FUNCTION_BLOCK TWO_POS_AXIS (* Composite Function Block Type *)
  (* Standard: 61499-2 *)
  (* Version 0.0, 4/29/2023, Dmitrii, Flexbridge AB, template *)
  PACKAGE UAO.Hackathon;
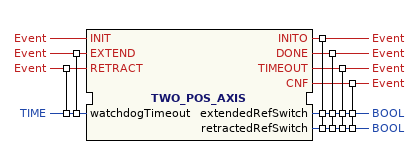
  EVENT_INPUT
    INIT; (* Initialization Request *)
    EXTEND WITH watchdogTimeout; (* Normal Execution Request *)
    RETRACT WITH watchdogTimeout;
  END_EVENT
  EVENT_OUTPUT
    INITO WITH extendedRefSwitch, retractedRefSwitch; (* Initialization Confirm *)
    DONE WITH retractedRefSwitch, extendedRefSwitch; (* Execution Confirmation *)
    TIMEOUT WITH retractedRefSwitch, extendedRefSwitch;
    CNF WITH extendedRefSwitch, retractedRefSwitch; (* Confirmation of an explicit or implicit data read request *)
  END_EVENT
  VAR_INPUT
    watchdogTimeout : TIME; (* Delay Time *)
  END_VAR
  VAR_OUTPUT
    extendedRefSwitch : BOOL; (* Current value(i) in the named variable array element *)
    retractedRefSwitch : BOOL; (* Current value(i) in the named variable array element *)
  END_VAR
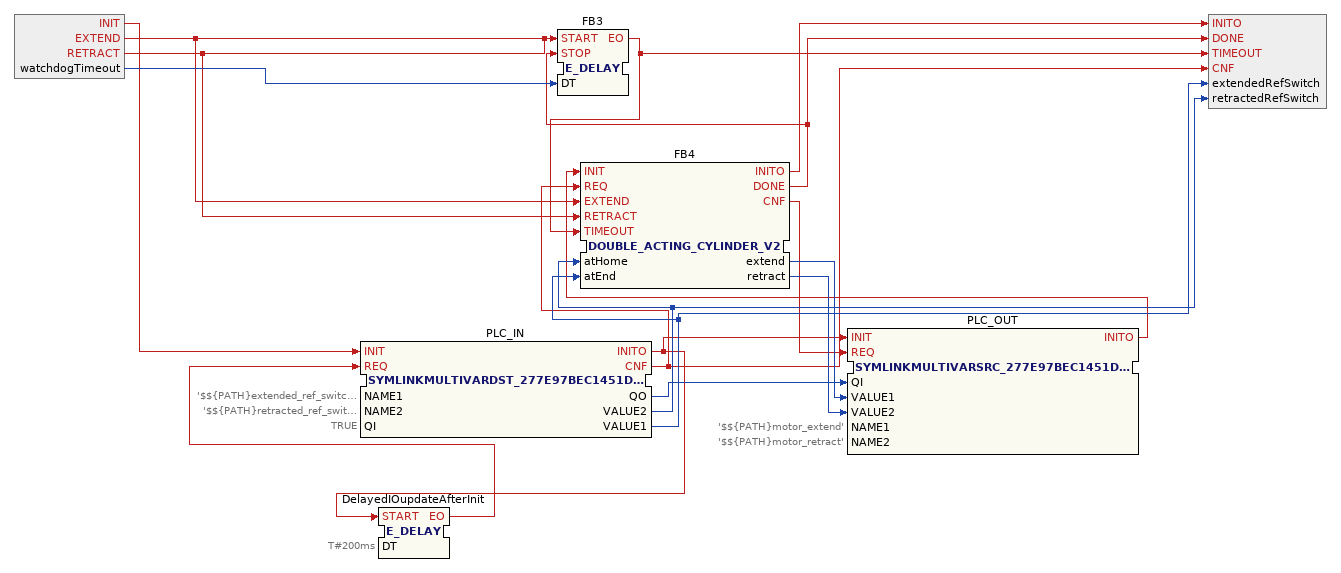
  FBS
    PLC_IN : SYMLINKMULTIVARDST_277E97BEC1451D2C(NAME1 := '$${PATH}extended_ref_switch', NAME2 := '$${PATH}retracted_ref_switch', QI := TRUE); {SET_ATTRIBUTE(Configuration.GenericFBType.InterfaceParams, Runtime.System#I:=2;VALUE${I$}:BOOL,BOOL)}
    PLC_OUT : SYMLINKMULTIVARSRC_277E97BEC1451D2C(NAME1 := '$${PATH}motor_extend', NAME2 := '$${PATH}motor_retract'); {SET_ATTRIBUTE(Configuration.GenericFBType.InterfaceParams, Runtime.System#I:=2;VALUE${I$}:BOOL,BOOL)}
    FB3 : E_DELAY;
    FB4 : DOUBLE_ACTING_CYLINDER_V2;
    DelayedIOupdateAfterInit : E_DELAY(DT := T#200ms);
  END_FBS
  EVENT_CONNECTIONS
    INIT TO PLC_IN.INIT;
    PLC_IN.INITO TO PLC_OUT.INIT;
    EXTEND TO FB3.START;
    RETRACT TO FB3.START;
    FB3.EO TO TIMEOUT;
    PLC_OUT.INITO TO FB4.INIT;
    FB4.INITO TO INITO;
    FB3.EO TO FB4.TIMEOUT;
    EXTEND TO FB4.EXTEND;
    RETRACT TO FB4.RETRACT;
    PLC_IN.CNF TO FB4.REQ;
    FB4.CNF TO PLC_OUT.REQ;
    FB4.DONE TO DONE;
    FB4.DONE TO FB3.STOP;
    PLC_IN.INITO TO DelayedIOupdateAfterInit.START;
    DelayedIOupdateAfterInit.EO TO PLC_IN.REQ;
    PLC_IN.CNF TO CNF;
  END_CONNECTIONS
  DATA_CONNECTIONS
    PLC_IN.QO TO PLC_OUT.QI;
    watchdogTimeout TO FB3.DT;
    FB4.extend TO PLC_OUT.VALUE1;
    FB4.retract TO PLC_OUT.VALUE2;
    PLC_IN.VALUE2 TO FB4.atHome;
    PLC_IN.VALUE1 TO FB4.atEnd;
    PLC_IN.VALUE1 TO extendedRefSwitch;
    PLC_IN.VALUE2 TO retractedRefSwitch;
  END_CONNECTIONS
END_FUNCTION_BLOCK
